(* IEC 61131-3 sources: programs/VI-54/VI-54_20171205/VI-54_20171205/Stations/Screen/LseClass170718/Class/Diagnostic, 1 file *)

(* ---- Diagnostic.st ---- *)
(*!
<Class
	Name               = "Diagnostic"
	Revision           = "1.0"
	RealtimeTask       = "false"
	CyclicTask         = "false"
	BackgroundTask     = "true"
	Sigmatek           = "false"
	OSInterface        = "false"
	HighPriority       = "false"
	Automatic          = "false"
	UpdateMode         = "Prescan"
	SharedCommandTable = "true"
	Objectsize         = "(630,360)">
	<Channels>
	</Channels>
	<RevDoku>
		<Owner Company="Sigmatek"/>
		<Dokumentation Revision="1.0" Date="2016-06-02" Author="HötAnt" Company="Sigmatek" Description="Creation"/>
	</RevDoku>
	<Network Name="Diagnostic">
		<!-- List of Components in this network -->
		<Components>
			<Object
				Name       = "_base"
				Class      = "DiagnosticBase"
				Position   = "(218,120)"
				Visualized = "false">
				<Channels>
					<Server Name="sLogError"/>
					<Server Name="sProgress"/>
					<Server Name="sStartExport"/>
					<Server Name="sStatus"/>
					<Server Name="sTraceError"/>
					<Client Name="cDriveLetter"/>
					<Client Name="cFileSys"/>
					<Client Name="cSigCLib"/>
					<Client Name="cSystemLogging"/>
				</Channels>
			</Object>
		</Components>
		<Comments>
		</Comments>
		<!-- List of Connections in this network -->
		<Connections>
			<Connection Source="this.sStatus" Destination="_base.sStatus" Vertices="(690,210),(518,210),"/>
			<Connection Source="this.sStartExport" Destination="_base.sStartExport" Vertices="(690,270),(518,270),"/>
			<Connection Source="this.sProgress" Destination="_base.sProgress" Vertices="(690,330),(518,330),"/>
			<Connection Source="this.sTraceError" Destination="_base.sTraceError" Vertices="(690,390),(518,390),"/>
			<Connection Source="_base.cSystemLogging" Destination="this.cSystemLogging" Vertices="(218,270),(38,210),"/>
			<Connection Source="this.sLogError" Destination="_base.sLogError" Vertices="(690,450),(518,450),"/>
			<Connection Source="_base.cDriveLetter" Destination="this.cDriveLetter" Vertices="(218,330),(38,270),"/>
		</Connections>
		<!-- Headerfiles -->
		<Options>
		</Options>
	</Network>
</Class>
*)
#pragma using DiagnosticBase

Diagnostic : CLASS
: DiagnosticBase
  //Servers:
  //Clients:
  //Variables:
  //Functions:
  //Tables:
	FUNCTION @STD
		VAR_OUTPUT
			ret_code	: CONFSTATES;
		END_VAR;
	FUNCTION GLOBAL TAB @CT_;
END_CLASS;
